FUNCTION_BLOCK TemperatureSensorScalingHandler
VAR_INPUT
	upperTemperatureSensor : INT;
	lowerTemperatureSensor : INT;
END_VAR
VAR_OUTPUT
	upperTemperatureValue : INT;
	lowerTemperatureValue : INT;
END_VAR
VAR
END_VAR


upperTemperatureValue	:= upperTemperatureSensor/10;
lowerTemperatureValue := lowerTemperatureSensor/10;

END_FUNCTION_BLOCK

(* stored: Version 1.1.0.1, ProductVersion 3.1.4024.9
   POU TemperatureSensorScalingHandler: Id {be2e305c-747a-4b45-b914-00c80fe2f05c}, SpecialFunc None *)
